(* IEC 61131-3 sources: volt/packages/volt-lsp-iec/test-corpus/lenze-mid/Device/Plc Logic/Application/A71_LocalSources/General, 8 files *)

(* ---- ATD_SR.pou ---- *)
FUNCTION ATD_SR : bool
VAR_INPUT
	iSet:BOOL;
	iReset: BOOL;
END_VAR
VAR
END_VAR
VAR_IN_OUT
	ioSR_value: BOOL;
END_VAR
%LANGUAGE ST

ioSR_value S=iSet;
ioSR_value R=iReset;

END_FUNCTION

(* ---- fc_DintToTime.pou ---- *)
FUNCTION fc_DintToTime : time
VAR_INPUT
	DintTime: DINT;
	DecShift: DINT :=0;
END_VAR
VAR
END_VAR

%LANGUAGE ST

fc_DintToTime:=DINT_TO_TIME(DintTime*1000/REAL_TO_DINT(EXPT(10,DecShift)));

END_FUNCTION

(* ---- RPM_To_DriveSpeed.pou ---- *)
FUNCTION RPM_To_DriveSpeed : bool
VAR_INPUT
	iEN: BOOL;
	iRPM: INT;
END_VAR
VAR
END_VAR
VAR_OUTPUT
	oDriveSpeed: INT;
END_VAR
%LANGUAGE LD
%NETWORK
MUL(EN := RAIL(), iRPM, 6, OUT => oDriveSpeed);

END_FUNCTION

(* ---- Bools_To_Byte.pou ---- *)
FUNCTION_BLOCK Bools_To_Byte
VAR
start1: POINTER TO BOOL;

i: USINT;
len: USINT;
byteval: BYTE;
END_VAR
VAR_INPUT
	adr_bit0_Of_Byte: POINTER TO bool;
END_VAR
VAR_OUTPUT
	oByte: BYTE;
END_VAR

%LANGUAGE ST
len:=7;
oByte:=0;

start1:= adr_bit0_Of_Byte;
oByte.0:= BOOL_TO_BIT(start1^);

start1:=adr_bit0_Of_Byte+1;
oByte.1:= BOOL_TO_BIT(start1^);

start1:=adr_bit0_Of_Byte+2;
oByte.2:= BOOL_TO_BIT(start1^);

start1:=adr_bit0_Of_Byte+3;
oByte.3:= BOOL_TO_BIT(start1^);

start1:=adr_bit0_Of_Byte+4;
oByte.4:= BOOL_TO_BIT(start1^);

start1:=adr_bit0_Of_Byte+5;
oByte.5:= BOOL_TO_BIT(start1^);

start1:=adr_bit0_Of_Byte+6;
oByte.6:= BOOL_TO_BIT(start1^);

start1:=adr_bit0_Of_Byte+7;
oByte.7:= BOOL_TO_BIT(start1^);

END_FUNCTION_BLOCK

(* ---- Byte_To_Bools.pou ---- *)
FUNCTION_BLOCK Byte_To_Bools
VAR
start1: POINTER TO BOOL;

i: USINT;
len: USINT;
tempByte: BYTE;
END_VAR
VAR_INPUT
	adr_bit0_Of_Byte: POINTER TO BOOL;
END_VAR
VAR_OUTPUT
	oByte: BYTE;
END_VAR

%LANGUAGE ST
len:=7;
oByte:=0;

start1:= adr_bit0_Of_Byte;

FOR i := 0 TO len DO
	tempByte:=REAL_TO_BYTE(EXPT(2,i));
    start1^:= BYTE_TO_BOOL((oByte AND tempByte)/tempByte);
END_FOR

END_FUNCTION_BLOCK

(* ---- GeneralMachineFlags.pou ---- *)
FUNCTION_BLOCK GeneralMachineFlags
VAR_INPUT
	iStartResetSeparate:BOOL;
	iServiceButtonHasResetFunction:BOOL;
	iFirstCycle:BOOL;
	iSignalPulse:BOOL;
	iAirPressureDoorsSeparate:BOOL;
	iEmergencyUnitOK:BOOL;
	iDoorUnitOK:BOOL;
	iSTO_Enabled:BOOL;
	iAirPressureOK:BOOL;
	iSwitchService:BOOL;
	iButtonService:BOOL;
	iStart1:BOOL;
	iStop1:BOOL;
	iReset1:BOOL;
	iAutoManual1:BOOL;
	iStart2:BOOL;
	iStop2:BOOL;
	iReset2:BOOL;
	iAutoManual2:BOOL;
	iStart3:BOOL;
	iStop3:BOOL;
	iReset3:BOOL;
	iAutoManual3:BOOL;
	iPreDelayAfterEmergStop: TIME;
	iPreStartDelayAuxDrives: TIME;
	iPreStopDelayAuxDrives: TIME;
	iPreDelayAfterSTOEnabled: TIME;

END_VAR
VAR_OUTPUT
	oResetEmergencyUnit:BOOL;
	oResetDoorUnit:BOOL;
	oStart1:BOOL;
	oStop1:BOOL;
	oReset1:BOOL;
	oCrossingDoorCircuit1:BOOL;
	oStart2:BOOL;
	oStop2:BOOL;
	oReset2:BOOL;
	oCrossingDoorCircuit2:BOOL;
	oStart3:BOOL;
	oStop3:BOOL;
	oReset3:BOOL;
	oCrossingDoorCircuit3:BOOL;
	oAlarm:BOOL;

END_VAR
VAR_IN_OUT
	GenFlags	: UDT_GeneralFlags;
END_VAR
VAR
	OneShotStart1: R_TRIG;
	OneShotStart2: R_TRIG;
	OneShotReset1: R_TRIG;
	OneShotReset2: BOOL;
	DnStartDelayAuxDrives: BOOL;
	DnStopDelayAuxDrives: BOOL;
	DnManualStopAuxDrives: BOOL;

	OffDelayPneumPressurised: TOF;
	OffDelayPneumSafetyGuard: TOF;
	OffDelayPneumEStop: TOF;

	OnDelayAfterEmergencyStop: TON;
	OnDelayStopAuxDrives: TON;
	OnDelayAfterSTOEnabled: TON;
	OnDelayManStopAuxDrives: TON;
	OnDelayStartAuxDrives: TON;

	RunAuto: SR;

END_VAR

%LANGUAGE LD
%NETWORK "NETWORK 2: Startup delay after emergency stop"
ASSIGN(OnDelayAfterEmergencyStop(IN := INVERT(iFirstCycle) AND iEmergencyUnitOK, PT := iPreDelayAfterEmergStop), Q => GenFlags.DelayAfterEmergStop);
%NETWORK "NETWORK 3: Startup delay after STO has been enabled"
ASSIGN(OnDelayAfterSTOEnabled(IN := GenFlags.DelayAfterEmergStop AND iSTO_Enabled, PT := iPreDelayAfterSTOEnabled), Q => GenFlags.DelayAfterSTO);
%NETWORK "NETWORK 4: Stop delay auxiliary drives"
VAR w1 : ANY; END_VAR
w1 := GenFlags.EnableAuxDrive AND INVERT(GenFlags.StartFlag) AND DnStartDelayAuxDrives AND INVERT(GenFlags.DriveIsRunning) AND INVERT(GenFlags.Rotflag);
ASSIGN(OnDelayStopAuxDrives(IN := w1, PT := iPreStopDelayAuxDrives), Q => DnStopDelayAuxDrives);
ASSIGN(BRANCH_SHORTCIRCUIT(FEED := w1, EQ(EN := RAIL(), iPreStopDelayAuxDrives, T#0MS).OUT, DnStopDelayAuxDrives), Q => DnStopDelayAuxDrives);
%NETWORK "NETWORK 5: Manual stop auxiliary drives"
ASSIGN(OnDelayManStopAuxDrives(IN := GenFlags.EnableAuxDrive AND (INVERT(iStop1) OR INVERT(iStop2) OR INVERT(iStop3)), PT := T#2S), Q => DnManualStopAuxDrives);
%NETWORK "NETWORK 6: Startup delay auxiliary drives"
VAR w2 : ANY; w3 : ANY; END_VAR
w2 := True;
w3 := w2 AND GenFlags.EnableAuxDrive AND INVERT(GenFlags.AuxDrivesStarted);
ASSIGN(OnDelayStartAuxDrives(IN := w3, PT := iPreStartDelayAuxDrives), Q => DnStartDelayAuxDrives);
ASSIGN(BRANCH_SHORTCIRCUIT(FEED := w3, EQ(EN := RAIL(), iPreStartDelayAuxDrives, T#0MS).OUT, DnStartDelayAuxDrives), Q => DnStartDelayAuxDrives);
ASSIGN(w2, Q_RESET => GenFlags.AuxDrivesStarted);
%NETWORK "NETWORK 7: Enable markers"
VAR w4 : ANY; w5 : ANY; END_VAR
w4 := GenFlags.DelayAfterEmergStop AND INVERT(GenFlags.MajorAlarm);
w5 := w4 AND iDoorUnitOK;
ASSIGN(w5 AND INVERT(GenFlags.DisableControl), Q => GenFlags.EnableControl);
ASSIGN(w5 AND GenFlags.EnableAuxDrive AND INVERT(GenFlags.AuxDrivesStarted) AND DnStartDelayAuxDrives, Q => GenFlags.EnableMainDrive);
ASSIGN(w4 AND (GenFlags.StartFlag OR GenFlags.RunAuto AND GenFlags.RestartAuxDrives OR GenFlags.EnableAuxDrive AND INVERT(DnStopDelayAuxDrives) AND INVERT(DnManualStopAuxDrives)), Q => GenFlags.EnableAuxDrive);
%NETWORK "NETWORK 8: Pneumatic markers"
VAR w6 : ANY; w7 : ANY; END_VAR
w6 := iEmergencyUnitOK;
ASSIGN(OffDelayPneumEStop(IN := w6, PT := T#1S), Q => GenFlags.EnablePneumEStop);
w7 := w6 AND (iSTO_Enabled OR INVERT(iAirPressureDoorsSeparate));
ASSIGN(OffDelayPneumSafetyGuard(IN := w7, PT := T#1S), Q => GenFlags.EnablePneumSafetyGuard);
ASSIGN(OffDelayPneumPressurised(IN := w7 AND iAirPressureOK, PT := T#1S), Q => GenFlags.EnablePneumPressurised);
%NETWORK "NETWORK 9: Active control panel"
VAR w8 : ANY; w9 : ANY; w10 : ANY; w11 : ANY; END_VAR
w8 := True;
ASSIGN(w8 AND iSwitchService, Q => GenFlags.ControlService);
w9 := w8 AND INVERT(iSwitchService);
ASSIGN(w9 AND iAutoManual1 AND INVERT(iAutoManual2) AND INVERT(iAutoManual3), Q => GenFlags.ControlMan1);
w10 := w9 AND INVERT(iAutoManual1);
ASSIGN(w10 AND iAutoManual2 AND INVERT(iAutoManual3), Q => GenFlags.ControlMan2);
w11 := w10 AND INVERT(iAutoManual2);
ASSIGN(w11 AND iAutoManual3, Q => GenFlags.ControlMan3);
ASSIGN(w11 AND INVERT(iAutoManual3), Q => GenFlags.ControlAuto);
%NETWORK "NETWORK 10: Control manual"
ASSIGN(GenFlags.EnableControl AND (GenFlags.ControlService AND iButtonService OR GenFlags.ControlMan1 AND iStart1 OR GenFlags.ControlMan2 AND iStart2 OR GenFlags.ControlMan3 AND iStart3) AND iStop1 AND iStop2 AND iStop3, Q => GenFlags.RunMan);
%NETWORK "NETWORK 11: Control automatic"
ASSIGN(RunAuto(SET1 := GenFlags.EnableControl AND GenFlags.ControlAuto AND (iStart1 OR iStart2 OR iStart3) AND iStop1 AND iStop2 AND iStop3, RESET := GenFlags.RunAuto AND (INVERT(GenFlags.EnableControl) OR INVERT(GenFlags.ControlAuto) OR INVERT(iStop1) OR INVERT(iStop2) OR INVERT(iStop3) OR INVERT(GenFlags.DriveIsRunning) AND (GenFlags.MinorAlarm OR GenFlags.MajorAlarm))), Q => GenFlags.RunAuto);
%NETWORK "DONE NETWORK 12: Start pulse"
ASSIGN(OneShotStart1(CLK := GenFlags.ControlService AND iButtonService OR GenFlags.ControlMan1 AND iStart1 OR GenFlags.ControlMan2 AND iStart2 OR GenFlags.ControlMan3 AND iStart3 OR GenFlags.ControlAuto AND (iStart1 OR iStart2 OR iStart3) OR OneShotStart2.Q) AND iStop1 AND iStop2 AND iStop3 OR OneShotStart2(CLK := GenFlags.RunMan OR GenFlags.RunAuto), Q => GenFlags.StartFlag);
%NETWORK "DONE NETWORK 13: Reset pulse"
ASSIGN(OneShotReset1(CLK := GenFlags.ControlService AND (iServiceButtonHasResetFunction AND iButtonService OR iReset1 OR iReset2 OR iReset3) OR (GenFlags.ControlMan1 OR GenFlags.ControlMan2 OR GenFlags.ControlMan3 OR GenFlags.ControlAuto) AND (iReset1 OR iReset2 OR iReset3)) AND iStop1 AND iStop2 AND iStop3 OR INVERT(iStartResetSeparate) AND GenFlags.StartFlag, Q => GenFlags.ResetFlag);
%NETWORK "DONE NETWORK 14: Stop flag"
ASSIGN(INVERT(iStop1) OR INVERT(iStop2) OR INVERT(iStop3) OR GenFlags.StopFlag AND INVERT(GenFlags.StartFlag), Q => GenFlags.StopFlag);
%NETWORK "DONE NETWORK 15: Reset safety unit"
ASSIGN((INVERT(iEmergencyUnitOK) OR iEmergencyUnitOK AND INVERT(iDoorUnitOK)) AND (iStartResetSeparate AND ((GenFlags.ControlMan1 OR GenFlags.ControlMan2 OR GenFlags.ControlMan3 OR GenFlags.ControlAuto) AND (iReset1 OR iReset2 OR iReset3) OR GenFlags.ControlService AND (iServiceButtonHasResetFunction AND iButtonService OR iReset1 OR iReset2 OR iReset3)) OR INVERT(iStartResetSeparate) AND ((GenFlags.ControlMan1 OR GenFlags.ControlAuto) AND iStart1 OR (GenFlags.ControlMan2 OR GenFlags.ControlAuto) AND iStart2 OR (GenFlags.ControlMan3 OR GenFlags.ControlAuto) AND iStart3 OR GenFlags.ControlService AND iButtonService) AND iStop1 AND iStop2 AND iStop3), Q => oResetEmergencyUnit);
%NETWORK "DONE NETWORK 16: Reset door unit"
ASSIGN(iEmergencyUnitOK AND INVERT(iDoorUnitOK) AND (iStartResetSeparate AND ((GenFlags.ControlMan1 OR GenFlags.ControlMan2 OR GenFlags.ControlMan3 OR GenFlags.ControlAuto) AND (iReset1 OR iReset2 OR iReset3) OR GenFlags.ControlService AND (iServiceButtonHasResetFunction AND iButtonService OR iReset1 OR iReset2 OR iReset3)) OR INVERT(iStartResetSeparate) AND ((GenFlags.ControlMan1 OR GenFlags.ControlAuto) AND iStart1 OR (GenFlags.ControlMan2 OR GenFlags.ControlAuto) AND iStart2 OR (GenFlags.ControlMan3 OR GenFlags.ControlAuto) AND iStart3 OR GenFlags.ControlService AND iButtonService) AND iStop1 AND iStop2 AND iStop3), Q => oResetDoorUnit);
%NETWORK "DONE NETWORK 17: Crossing doorcircuit control panel 1"
ASSIGN(GenFlags.ControlMan1, Q => oCrossingDoorCircuit1);
%NETWORK "DONE NETWORK 18: Crossing doorcircuit control panel 2"
ASSIGN(GenFlags.ControlMan2, Q => oCrossingDoorCircuit2);
%NETWORK "DONE NETWORK 19: Crossing doorcircuit control panel 3"
ASSIGN(GenFlags.ControlMan3, Q => oCrossingDoorCircuit3);
%NETWORK "DONE NETWORK 20: Signal lamps control panel 1 "
VAR w12 : ANY; END_VAR
w12 := True;
ASSIGN(w12 AND (GenFlags.ControlMan1 OR GenFlags.ControlAuto) AND ((GenFlags.RunMan OR GenFlags.RunAuto) AND INVERT(GenFlags.MinorAlarm) AND INVERT(GenFlags.MajorAlarm) OR (GenFlags.EnableControl OR INVERT(iStartResetSeparate) AND (GenFlags.MinorAlarm OR GenFlags.MajorAlarm)) AND iSignalPulse AND (INVERT(GenFlags.MinorAlarm) AND INVERT(GenFlags.MajorAlarm) OR INVERT(iStartResetSeparate))), Q => oStart1);
ASSIGN(w12 AND iEmergencyUnitOK AND (INVERT(GenFlags.RunMan) OR INVERT(GenFlags.ControlMan1)) AND INVERT(GenFlags.RunAuto), Q => oStop1);
ASSIGN(w12 AND (GenFlags.ControlMan1 OR GenFlags.ControlMan2 OR GenFlags.ControlMan3 OR GenFlags.ControlAuto OR GenFlags.ControlService) AND (GenFlags.MinorAlarm OR GenFlags.MajorAlarm OR INVERT(iDoorUnitOK)) AND iSignalPulse, Q => oReset1);
%NETWORK "DONE NETWORK 21: Signal lamps control panel 2"
VAR w13 : ANY; END_VAR
w13 := True;
ASSIGN(w13 AND (GenFlags.ControlMan2 OR GenFlags.ControlAuto) AND ((GenFlags.RunMan OR GenFlags.RunAuto) AND INVERT(GenFlags.MinorAlarm) AND INVERT(GenFlags.MajorAlarm) OR (GenFlags.EnableControl OR INVERT(iStartResetSeparate) AND (GenFlags.MinorAlarm OR GenFlags.MajorAlarm)) AND iSignalPulse AND (INVERT(GenFlags.MinorAlarm) AND INVERT(GenFlags.MajorAlarm) OR INVERT(iStartResetSeparate))), Q => oStart2);
ASSIGN(w13 AND iEmergencyUnitOK AND (INVERT(GenFlags.RunMan) OR INVERT(GenFlags.ControlMan1)) AND INVERT(GenFlags.RunAuto), Q => oStop2);
ASSIGN(w13 AND (GenFlags.ControlMan1 OR GenFlags.ControlMan2 OR GenFlags.ControlMan3 OR GenFlags.ControlAuto OR GenFlags.ControlService) AND (GenFlags.MinorAlarm OR GenFlags.MajorAlarm OR INVERT(iDoorUnitOK)) AND iSignalPulse, Q => oReset2);
%NETWORK "DONE NETWORK 22: Signal lamps control panel 3"
VAR w14 : ANY; END_VAR
w14 := True;
ASSIGN(w14 AND (GenFlags.ControlMan3 OR GenFlags.ControlAuto) AND ((GenFlags.RunMan OR GenFlags.RunAuto) AND INVERT(GenFlags.MinorAlarm) AND INVERT(GenFlags.MajorAlarm) OR (GenFlags.EnableControl OR INVERT(iStartResetSeparate) AND (GenFlags.MinorAlarm OR GenFlags.MajorAlarm)) AND iSignalPulse AND (INVERT(GenFlags.MinorAlarm) AND INVERT(GenFlags.MajorAlarm) OR INVERT(iStartResetSeparate))), Q => oStart3);
ASSIGN(w14 AND iEmergencyUnitOK AND (INVERT(GenFlags.RunMan) OR INVERT(GenFlags.ControlMan1)) AND INVERT(GenFlags.RunAuto), Q => oStop3);
ASSIGN(w14 AND (GenFlags.ControlMan1 OR GenFlags.ControlMan2 OR GenFlags.ControlMan3 OR GenFlags.ControlAuto OR GenFlags.ControlService) AND (GenFlags.MinorAlarm OR GenFlags.MajorAlarm OR INVERT(iDoorUnitOK)) AND iSignalPulse, Q => oReset3);
%NETWORK "TODO NETWORK 23: Signal lamp alarm"
ASSIGN((GenFlags.Warning OR GenFlags.MinorAlarm OR GenFlags.MajorAlarm) AND iSignalPulse, Q => oAlarm);
%NETWORK "DONE NETWORK 24: Only when during a complete CPU cycle there is no alarm, the $"Active$"-alarm signals are reset"
VAR w15 : ANY; END_VAR
w15 := True;
ASSIGN(w15 AND GenFlags.Warning, Q => GenFlags.WarningActive);
ASSIGN(w15 AND GenFlags.MinorAlarm, Q => GenFlags.MinorAlarmActive);
ASSIGN(w15 AND GenFlags.MajorAlarm, Q => GenFlags.MajorAlarmActive);
%NETWORK "DONE NETWORK 25: Reset alarm actions"
ASSIGN(True, Q_RESET => GenFlags.Warning, Q_RESET => GenFlags.MinorAlarm, Q_RESET => GenFlags.MajorAlarm, Q_RESET => GenFlags.DummyWarning, Q_RESET => GenFlags.DisableControl);
%NETWORK "TODO NETWORK 26: SAVE"

END_FUNCTION_BLOCK

(* ---- GeneralProgramFlags.pou ---- *)
PROGRAM GeneralProgramFlags
VAR_INPUT
END_VAR
VAR_OUTPUT
END_VAR
VAR
	AlwaysOff: BOOL;
	AlwaysOn: BOOL;
	OS: BOOL;
	first: BOOL;
	flag: BOOL;
	OSfirstflagcycle: BOOL;
	FirstCycle: BOOL;
	dummyWord: INT;
	tmr_FF500ms: TON;
	tmr_FF500ms_not: TON;
	tmr_FF100ms: TON;
	tmr_FF100ms_not: TON;
	tmr_FF50ms: TON;
	tmr_FF50ms_not: TON;
	tmr_FF1s: TON;
	tmr_FF1s_not: TON;
	PLC_StartUp_Delay: TON;
END_VAR

%LANGUAGE LD
%NETWORK
// Always Off
ASSIGN(AlwaysOff, Q_RESET => AlwaysOff);
%NETWORK
// Always ON
ASSIGN(INVERT(AlwaysOn), Q_SET => AlwaysOn);
%NETWORK
ASSIGN(AlwaysOn AND OSfirstflagcycle, Q_RESET => FirstCycle);
%NETWORK
MOVE(EN := AlwaysOn, 0, OUT => dummyWord);
%NETWORK
VAR w1 : ANY; END_VAR
w1 := RAIL();
ASSIGN(tmr_FF50ms(IN := w1 AND INVERT(tmr_FF50ms_not.Q), PT := T#100MS), Q => FF50ms);
ASSIGN(tmr_FF50ms_not(IN := w1 AND FF50ms, PT := T#100MS), Q => LST_General.Imp100ms);
%NETWORK
VAR w2 : ANY; END_VAR
w2 := RAIL();
ASSIGN(tmr_FF100ms(IN := w2 AND INVERT(tmr_FF100ms_not.Q), PT := T#500MS), Q => FF100ms);
ASSIGN(tmr_FF100ms_not(IN := w2 AND FF100ms, PT := T#500MS), Q => LST_General.Imp200ms);
%NETWORK
VAR w3 : ANY; END_VAR
w3 := RAIL();
ASSIGN(tmr_FF500ms(IN := w3 AND INVERT(tmr_FF500ms_not.Q), PT := T#500MS), Q => FF500ms);
ASSIGN(tmr_FF500ms_not(IN := w3 AND FF500ms, PT := T#500MS), Q => LST_General.Imp1s);
%NETWORK
VAR w4 : ANY; END_VAR
w4 := RAIL();
ASSIGN(tmr_FF1s(IN := w4 AND INVERT(tmr_FF1s_not.Q), PT := T#1S), Q => FF1s);
tmr_FF1s_not(IN := w4 AND FF1s, PT := T#1S);
%NETWORK
ASSIGN(PLC_StartUp_Delay(IN := AlwaysOn, PT := T#60S), Q => LST_General.StartUpDelayPLC);

END_PROGRAM

(* ---- Simulation.pou ---- *)
PROGRAM Simulation
VAR
	ATD_Simulate: BOOL;
END_VAR

%LANGUAGE ST
IF (ATD_Simulate) THEN
Mach1_Safety.Status.Emergency_button01:=TRUE;
Mach1_Safety.Status.Emergency_button02:=TRUE;
Mach1_Safety.Status.Emergency_button03:=TRUE;
Mach1_Safety.Status.Emergency_button04:=TRUE;
Mach1_Safety.Status.Emergency_button05:=TRUE;
Mach1_Safety.Status.EmergencyStopOK :=TRUE;

LST_InputsOutputs.I100_2_Pushbutton_stop_OP0a:=TRUE;
LST_InputsOutputs.I132_2_PB_Stop_OP2a :=TRUE;
LST_InputsOutputs.I100_0_AirpressureOK:=TRUE;
LST_InputsOutputs.I100_3_Selector_switch_auto_manual_OP0a:=FALSE;
LST_InputsOutputs.I100_1_Pushbutton_start_OP0a:=TRUE;

END_IF

END_PROGRAM
